// TIA Portal V16 export
// export: Created 2021-07-12T14:47:17.4795713Z, ExportSetting WithDefaults, DisplayName Totally Integrated Automation Portal, DisplayVersion V16, DisplayName TIA Portal Version Control Interface, DisplayVersion V16, DisplayName TIA Portal Openness, DisplayVersion V16, DisplayName STEP 7 Professional, DisplayVersion V16, DisplayName STEP 7 Safety, DisplayVersion V16, DisplayName WinCC Professional, DisplayVersion V16
VAR_GLOBAL   // PLC tag table "Default tag table"
   Tag_1 AT %M66.0 : Bool;
   Tag_2 AT %M60.0 : Bool;
   Tag_3 AT %M60.1 : Bool;
   Tag_4 AT %M60.2 : Bool;
   Tag_5 AT %M60.3 : Bool;
   Tag_6 AT %M70.0 : Bool;
   Tag_7 AT %M1.0 : Bool;
   Tag_8 AT %M1.1 : Bool;
   Tag_9 AT %M1.2 : Bool;
   Tag_10 AT %M70.1 : Bool;
   Tag_11 AT %M60.5 : Bool;
   Tag_12 AT %IW0 : Word;
   Tag_13 AT %IW2 : Word;
   Tag_14 AT %IW4 : Word;
   Tag_15 AT %M66.3 : Bool;
   Tag_16 AT %M17.0 : Bool;
   Tag_17 AT %M1717.0 : Bool;
   adım1 AT %M0.0 : Bool;
   step1 AT %M0.1 : Bool;
   step2 AT %M0.2 : Bool;
   step3 AT %M0.3 : Bool;
   step4 AT %M0.4 : Bool;
   step5 AT %M0.5 : Bool;
   Tag_18 AT %M170.0 : Bool;
   Tag_19 AT %M170.1 : Bool;
   step6 AT %M0.6 : Bool;
   step7 AT %M0.7 : Bool;
   Tag_20 AT %M1717.2 : Bool;
   Tag_21 AT %MD100 : DWord;
END_VAR
